RoboDK station: custom-palletizing.rdk

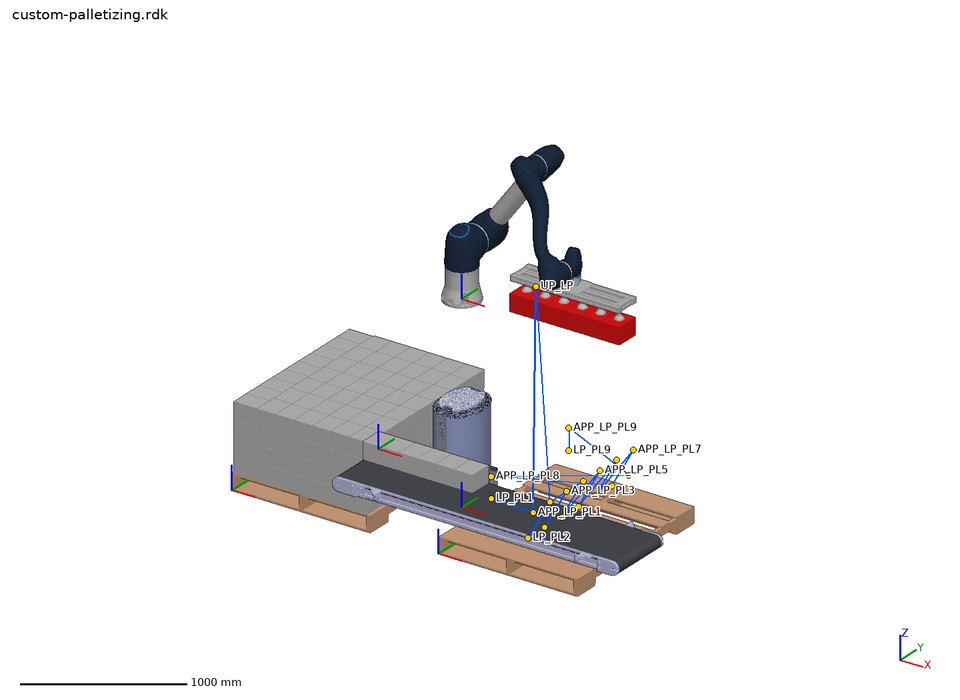
[picture v0: the station drawn from its stored meshes, robots at their saved joint values, targets as dots, program paths as lines]
Station custom-palletizing (saved by RoboDK 5.7.1). Poses are relative to the parent item; angles as X-Y-Z fixed-axis rotations.
Station parameters (name, value as stored): Conv_Run, 1
  - frame World at (0, 0, 0) mm
    - frame Doosan Robotics H2515 Base at (0, 0, 1390) mm
      - robot Doosan Robotics H2515: 6 axes, payload 25 kg, reach 1500 mm, repeatability 0.1 mm
          modified DH rows (alpha deg, a mm, theta deg, d mm): 0, 0, 0, 344.3; -90, 0, -90, -9.9; 0, 759.5, -90, 0; -90, 0, 0, 619.5; 90, 0, 0, 0; -90, 0, 0, 121
          base shift (0, 0, 0) mm, rotated rx 0 ry 0 rz 180 deg
          joint limits [-360, -130, -160, -360, -360, -360] to [360, 130, 160, 360, 360, 360]; home [0, 0, 90, 0, 0, 0]; saved at [0.72, 36.475, 109.267, -180, -34.248, -179.28]
        - tool Gripper, TCP at (0, 0, 145) mm, size 790 x 190 x 145 mm
          - object REF at (-402, -90, 0) mm, size 805 x 170 x 120 mm, geometry from 6 cajas.STEP
    - frame Conveyor_Frame at (0, -870, 737) mm
      - object Conveyor at (0, 300, -50) mm, size 2090.8 x 597 x 107.2 mm
      - object REF_CVY_BOX at (0, -170, 0) mm, size 805 x 170 x 120 mm, geometry from 6 cajas.STEP
      - folder Pick_poses
        - target APP_PICK (Cartesian target) at (402, -89.5, 320) mm, rotated rx 180 ry 0 rz 0 deg; joints [-67.813, 42.819, 79.411, 0, 57.77, 112.187] of Doosan Robotics H2515
        - target PICK_POSE (Cartesian target) at (402, -89.5, 120) mm, rotated rx -180 ry 0 rz 0 deg; joints [-67.813, 52.353, 82.536, 0, 45.111, 112.187] of Doosan Robotics H2515
        - target RET_PICK (Cartesian target) at (402, -89.5, 520) mm, rotated rx -180 ry 0 rz 0 deg; joints [-67.813, 36.264, 71.178, 0, 72.558, 112.187] of Doosan Robotics H2515
      - folder Pick_Aux_Poses
        - target UP_CONV (Cartesian target) at (402, 255, 850) mm, rotated rx -180 ry 0 rz 0 deg; joints [-57.601, 8.724, 80.723, 0, 90.554, 122.399] of Doosan Robotics H2515
    - frame Left_Pallet_Frame at (250, -600, 0) mm
      - object Left_Pallet at (0, 0, 0) mm, size 1016 x 1219.2 x 114.3 mm, geometry from Pallet-40x48in (1).sld
      - folder Ref_Box_LP
        - folder LAYER1
          - object REF_RP_BOX1 at (190, 0, 115) mm, size 805 x 170 x 120 mm, geometry from 6 cajas.STEP
          - object REF_RP_BOX2 at (190, 175, 115) mm, size 805 x 170 x 120 mm, geometry from 6 cajas.STEP
          - object REF_RP_BOX3 at (190, 350, 115) mm, size 805 x 170 x 120 mm, geometry from 6 cajas.STEP
          - object REF_RP_BOX4 at (190, 525, 115) mm, size 805 x 170 x 120 mm, geometry from 6 cajas.STEP
          - object REF_RP_BOX5 at (190, 700, 115) mm, size 805 x 170 x 120 mm, geometry from 6 cajas.STEP
          - object REF_RP_BOX6 at (190, 875, 115) mm, size 805 x 170 x 120 mm, geometry from 6 cajas.STEP
          - object REF_RP_BOX7 at (190, 1050, 115) mm, size 805 x 170 x 120 mm, geometry from 6 cajas.STEP
          - object REF_RP_BOX8 at (185, 0, 115) mm, rotated rx 0 ry 0 rz 90 deg, size 805 x 170 x 120 mm, geometry from 6 cajas.STEP
          - object REF_RP_BOX9 at (185, 810, 115) mm, rotated rx 0 ry 0 rz 90 deg, size 400 x 170 x 120 mm, geometry from 3 cajas.STEP
        - folder LAYER2
          - object REF_RP_BOX10 at (995, 815, 236) mm, rotated rx 0 ry 0 rz 90 deg, size 400 x 170 x 120 mm, geometry from 3 cajas.STEP
          - object REF_RP_BOX11 at (995, 5, 236) mm, rotated rx 0 ry 0 rz 90 deg, size 805 x 170 x 120 mm, geometry from 6 cajas.STEP
          - object REF_RP_BOX12 at (15, 0, 236) mm, size 805 x 170 x 120 mm, geometry from 6 cajas.STEP
          - object REF_RP_BOX13 at (15, 175, 236) mm, size 805 x 170 x 120 mm, geometry from 6 cajas.STEP
          - object REF_RP_BOX14 at (15, 350, 236) mm, size 805 x 170 x 120 mm, geometry from 6 cajas.STEP
          - object REF_RP_BOX15 at (15, 525, 236) mm, size 805 x 170 x 120 mm, geometry from 6 cajas.STEP
          - object REF_RP_BOX16 at (15, 700, 236) mm, size 805 x 170 x 120 mm, geometry from 6 cajas.STEP
          - object REF_RP_BOX17 at (15, 875, 236) mm, size 805 x 170 x 120 mm, geometry from 6 cajas.STEP
          - object REF_RP_BOX18 at (15, 1050, 236) mm, size 805 x 170 x 120 mm, geometry from 6 cajas.STEP
        - folder LAYER3
          - object REF_RP_BOX19 at (190, 0, 357) mm, size 805 x 170 x 120 mm, geometry from 6 cajas.STEP
          - object REF_RP_BOX20 at (190, 175, 357) mm, size 805 x 170 x 120 mm, geometry from 6 cajas.STEP
          - object REF_RP_BOX21 at (190, 350, 357) mm, size 805 x 170 x 120 mm, geometry from 6 cajas.STEP
          - object REF_RP_BOX22 at (190, 525, 357) mm, size 805 x 170 x 120 mm, geometry from 6 cajas.STEP
          - object REF_RP_BOX23 at (190, 700, 357) mm, size 805 x 170 x 120 mm, geometry from 6 cajas.STEP
          - object REF_RP_BOX24 at (190, 875, 357) mm, size 805 x 170 x 120 mm, geometry from 6 cajas.STEP
          - object REF_RP_BOX25 at (190, 1050, 357) mm, size 805 x 170 x 120 mm, geometry from 6 cajas.STEP
          - object REF_RP_BOX26 at (185, 0, 357) mm, rotated rx 0 ry 0 rz 90 deg, size 805 x 170 x 120 mm, geometry from 6 cajas.STEP
          - object REF_RP_BOX27 at (185, 810, 357) mm, rotated rx 0 ry 0 rz 90 deg, size 400 x 170 x 120 mm, geometry from 3 cajas.STEP
        - folder LAYER4
          - object REF_RP_BOX28 at (995, 815, 477) mm, rotated rx 0 ry 0 rz 90 deg, size 400 x 170 x 120 mm, geometry from 3 cajas.STEP
          - object REF_RP_BOX29 at (995, 5, 477) mm, rotated rx 0 ry 0 rz 90 deg, size 805 x 170 x 120 mm, geometry from 6 cajas.STEP
          - object REF_RP_BOX30 at (15, 0, 477) mm, size 805 x 170 x 120 mm, geometry from 6 cajas.STEP
          - object REF_RP_BOX31 at (15, 175, 477) mm, size 805 x 170 x 120 mm, geometry from 6 cajas.STEP
          - object REF_RP_BOX32 at (15, 350, 477) mm, size 805 x 170 x 120 mm, geometry from 6 cajas.STEP
          - object REF_RP_BOX33 at (15, 525, 477) mm, size 805 x 170 x 120 mm, geometry from 6 cajas.STEP
          - object REF_RP_BOX34 at (15, 700, 477) mm, size 805 x 170 x 120 mm, geometry from 6 cajas.STEP
          - object REF_RP_BOX35 at (15, 875, 477) mm, size 805 x 170 x 120 mm, geometry from 6 cajas.STEP
          - object REF_RP_BOX36 at (15, 1050, 477) mm, size 805 x 170 x 120 mm, geometry from 6 cajas.STEP
        - folder LAYER5
          - object REF_RP_BOX37 at (190, 0, 597) mm, size 805 x 170 x 120 mm, geometry from 6 cajas.STEP
          - object REF_RP_BOX38 at (190, 175, 597) mm, size 805 x 170 x 120 mm, geometry from 6 cajas.STEP
          - object REF_RP_BOX39 at (190, 350, 597) mm, size 805 x 170 x 120 mm, geometry from 6 cajas.STEP
          - object REF_RP_BOX40 at (190, 525, 597) mm, size 805 x 170 x 120 mm, geometry from 6 cajas.STEP
          - object REF_RP_BOX41 at (190, 700, 597) mm, size 805 x 170 x 120 mm, geometry from 6 cajas.STEP
          - object REF_RP_BOX42 at (190, 875, 597) mm, size 805 x 170 x 120 mm, geometry from 6 cajas.STEP
          - object REF_RP_BOX43 at (190, 1050, 597) mm, size 805 x 170 x 120 mm, geometry from 6 cajas.STEP
          - object REF_RP_BOX44 at (185, 0, 597) mm, rotated rx 0 ry 0 rz 90 deg, size 805 x 170 x 120 mm, geometry from 6 cajas.STEP
          - object REF_RP_BOX45 at (185, 810, 597) mm, rotated rx 0 ry 0 rz 90 deg, size 400 x 170 x 120 mm, geometry from 3 cajas.STEP
        - folder LAYER6
          - object REF_RP_BOX46 at (995, 815, 717) mm, rotated rx 0 ry 0 rz 90 deg, size 400 x 170 x 120 mm, geometry from 3 cajas.STEP
          - object REF_RP_BOX47 at (995, 5, 717) mm, rotated rx 0 ry 0 rz 90 deg, size 805 x 170 x 120 mm, geometry from 6 cajas.STEP
          - object REF_RP_BOX48 at (15, 0, 717) mm, size 805 x 170 x 120 mm, geometry from 6 cajas.STEP
          - object REF_RP_BOX49 at (15, 175, 717) mm, size 805 x 170 x 120 mm, geometry from 6 cajas.STEP
          - object REF_RP_BOX50 at (15, 350, 717) mm, size 805 x 170 x 120 mm, geometry from 6 cajas.STEP
          - object REF_RP_BOX51 at (15, 525, 717) mm, size 805 x 170 x 120 mm, geometry from 6 cajas.STEP
          - object REF_RP_BOX52 at (15, 700, 717) mm, size 805 x 170 x 120 mm, geometry from 6 cajas.STEP
          - object REF_RP_BOX53 at (15, 875, 717) mm, size 805 x 170 x 120 mm, geometry from 6 cajas.STEP
          - object REF_RP_BOX54 at (15, 1050, 717) mm, size 805 x 170 x 120 mm, geometry from 6 cajas.STEP
        - folder LAYER7
          - object REF_RP_BOX55 at (190, 0, 837) mm, size 805 x 170 x 120 mm, geometry from 6 cajas.STEP
          - object REF_RP_BOX56 at (190, 175, 837) mm, size 805 x 170 x 120 mm, geometry from 6 cajas.STEP
          - object REF_RP_BOX57 at (190, 350, 837) mm, size 805 x 170 x 120 mm, geometry from 6 cajas.STEP
          - object REF_RP_BOX58 at (190, 525, 837) mm, size 805 x 170 x 120 mm, geometry from 6 cajas.STEP
          - object REF_RP_BOX59 at (190, 700, 837) mm, size 805 x 170 x 120 mm, geometry from 6 cajas.STEP
          - object REF_RP_BOX60 at (190, 875, 837) mm, size 805 x 170 x 120 mm, geometry from 6 cajas.STEP
          - object REF_RP_BOX61 at (190, 1050, 837) mm, size 805 x 170 x 120 mm, geometry from 6 cajas.STEP
          - object REF_RP_BOX62 at (185, 0, 837) mm, rotated rx 0 ry 0 rz 90 deg, size 805 x 170 x 120 mm, geometry from 6 cajas.STEP
          - object REF_RP_BOX63 at (185, 810, 837) mm, rotated rx 0 ry 0 rz 90 deg, size 400 x 170 x 120 mm, geometry from 3 cajas.STEP
        - folder LAYER8
          - object REF_RP_BOX64 at (995, 815, 957) mm, rotated rx 0 ry 0 rz 90 deg, size 400 x 170 x 120 mm, geometry from 3 cajas.STEP
          - object REF_RP_BOX65 at (995, 5, 957) mm, rotated rx 0 ry 0 rz 90 deg, size 805 x 170 x 120 mm, geometry from 6 cajas.STEP
          - object REF_RP_BOX66 at (15, 0, 957) mm, size 805 x 170 x 120 mm, geometry from 6 cajas.STEP
          - object REF_RP_BOX67 at (15, 175, 957) mm, size 805 x 170 x 120 mm, geometry from 6 cajas.STEP
          - object REF_RP_BOX68 at (15, 350, 957) mm, size 805 x 170 x 120 mm, geometry from 6 cajas.STEP
          - object REF_RP_BOX69 at (15, 525, 957) mm, size 805 x 170 x 120 mm, geometry from 6 cajas.STEP
          - object REF_RP_BOX70 at (15, 700, 957) mm, size 805 x 170 x 120 mm, geometry from 6 cajas.STEP
          - object REF_RP_BOX71 at (15, 875, 957) mm, size 805 x 170 x 120 mm, geometry from 6 cajas.STEP
          - object REF_RP_BOX72 at (15, 1050, 957) mm, size 805 x 170 x 120 mm, geometry from 6 cajas.STEP
        - folder LAYER9
          - object REF_RP_BOX73 at (190, 0, 1077) mm, size 805 x 170 x 120 mm, geometry from 6 cajas.STEP
          - object REF_RP_BOX74 at (190, 175, 1077) mm, size 805 x 170 x 120 mm, geometry from 6 cajas.STEP
          - object REF_RP_BOX75 at (190, 350, 1077) mm, size 805 x 170 x 120 mm, geometry from 6 cajas.STEP
          - object REF_RP_BOX76 at (190, 525, 1077) mm, size 805 x 170 x 120 mm, geometry from 6 cajas.STEP
          - object REF_RP_BOX77 at (190, 700, 1077) mm, size 805 x 170 x 120 mm, geometry from 6 cajas.STEP
          - object REF_RP_BOX78 at (190, 875, 1077) mm, size 805 x 170 x 120 mm, geometry from 6 cajas.STEP
          - object REF_RP_BOX79 at (190, 1050, 1077) mm, size 805 x 170 x 120 mm, geometry from 6 cajas.STEP
          - object REF_RP_BOX80 at (185, 0, 1077) mm, rotated rx 0 ry 0 rz 90 deg, size 805 x 170 x 120 mm, geometry from 6 cajas.STEP
          - object REF_RP_BOX81 at (185, 810, 1077) mm, rotated rx 0 ry 0 rz 90 deg, size 400 x 170 x 120 mm, geometry from 3 cajas.STEP
      - folder LP_Aux_Poses
        - target UP_LP (Cartesian target) at (250, 660, 1590) mm, rotated rx 180 ry 0 rz 90 deg; joints [5.716, -8.781, 97.939, 0, 90.842, 95.716] of Doosan Robotics H2515
      - folder App_PL_LP
        - folder APP_LAYER 1
          - target APP_LP_PL1 (Cartesian target) at (593, 140, 385) mm, rotated rx -180 ry 0 rz -180 deg; joints [-29.211, 79.655, 80.222, 0, 20.123, -29.211] of Doosan Robotics H2515
          - target APP_LP_PL2 (Cartesian target) at (593, 315, 385) mm, rotated rx -180 ry 0 rz 180 deg; joints [-19.317, 78.101, 88.207, 0, 13.692, -19.317] of Doosan Robotics H2515
          - target APP_LP_PL3 (Cartesian target) at (593, 490, 385) mm, rotated rx -180 ry 0 rz -180 deg; joints [-8.102, 77.483, 92.417, 0, 10.1, -8.102] of Doosan Robotics H2515
          - target APP_LP_PL4 (Cartesian target) at (593, 665, 385) mm, rotated rx -180 ry 0 rz 180 deg; joints [3.738, 77.423, 92.897, 0, 9.68, 3.738] of Doosan Robotics H2515
          - target APP_LP_PL5 (Cartesian target) at (593, 840, 385) mm, rotated rx -180 ry 0 rz 180 deg; joints [15.244, 77.873, 89.645, 0, 12.482, 15.244] of Doosan Robotics H2515
          - target APP_LP_PL6 (Cartesian target) at (593, 1015, 385) mm, rotated rx -180 ry 0 rz -180 deg; joints [25.607, 79.136, 82.646, 0, 18.218, 25.607] of Doosan Robotics H2515
          - target APP_LP_PL7 (Cartesian target) at (593, 1190, 385) mm, rotated rx -180 ry 0 rz 180 deg; joints [34.436, 81.771, 71.646, 0, 26.584, 34.436] of Doosan Robotics H2515
          - target APP_LP_PL8 (Cartesian target) at (105, 402, 385) mm, rotated rx 180 ry 0 rz 90 deg; joints [-30.546, 85.041, 129.392, 0, -34.433, 59.454] of Doosan Robotics H2515
          - target APP_LP_PL9 (Cartesian target) at (105, 1212, 385) mm, rotated rx 180 ry 0 rz 90 deg; joints [59.082, 76.805, 106.157, 0, -2.962, 149.082] of Doosan Robotics H2515
        - folder APP_LAYER 2
          - target APP_LP_PL10 (Cartesian target) at (865, 812, 506) mm, rotated rx -180 ry 0 rz 90 deg; joints [9.768, 78.069, 62.913, 0, 39.018, 99.768] of Doosan Robotics H2515
          - target APP_LP_PL11 (Cartesian target) at (865, 407, 506) mm, rotated rx 180 ry 0 rz 90 deg; joints [-10.819, 78.078, 62.886, 0, 39.036, 79.181] of Doosan Robotics H2515
          - target APP_LP_PL12 (Cartesian target) at (418, 140, 506) mm, rotated rx 180 ry 0 rz 180 deg; joints [-35.824, 67.971, 101.551, 0, 10.478, -35.824] of Doosan Robotics H2515
          - target APP_LP_PL13 (Cartesian target) at (418, 315, 506) mm, rotated rx -180 ry 0 rz -180 deg; joints [-24.604, 67.188, 110.029, 0, 2.783, -24.604] of Doosan Robotics H2515
          - target APP_LP_PL14 (Cartesian target) at (418, 490, 506) mm, rotated rx -180 ry 0 rz -180 deg; joints [-11.02, 67.158, 114.814, 0, -1.972, -11.02] of Doosan Robotics H2515
          - target APP_LP_PL15 (Cartesian target) at (418, 665, 506) mm, rotated rx -180 ry 0 rz -180 deg; joints [3.861, 67.187, 115.58, 0, -2.766, 3.861] of Doosan Robotics H2515
          - target APP_LP_PL16 (Cartesian target) at (418, 840, 506) mm, rotated rx -180 ry 0 rz 180 deg; joints [18.196, 67.131, 112.257, 0, 0.612, 18.196] of Doosan Robotics H2515
          - target APP_LP_PL17 (Cartesian target) at (418, 1015, 506) mm, rotated rx 180 ry 0 rz 180 deg; joints [30.502, 67.544, 105.11, 0, 7.346, 30.502] of Doosan Robotics H2515
          - target APP_LP_PL18 (Cartesian target) at (418, 1190, 506) mm, rotated rx -180 ry 0 rz 180 deg; joints [40.325, 69.172, 94.445, 0, 16.383, 40.325] of Doosan Robotics H2515
        - folder APP_LAYER 3
          - target APP_LP_PL19 (Cartesian target) at (593, 140, 835) mm, rotated rx -180 ry 0 rz -180 deg; joints [-10.819, 78.078, 62.886, 0, 39.036, 79.181] of Doosan Robotics H2515
          - target APP_LP_PL20 (Cartesian target) at (593, 315, 835) mm, rotated rx -180 ry 0 rz 180 deg; joints [-10.819, 78.078, 62.886, 0, 39.036, 79.181] of Doosan Robotics H2515
          - target APP_LP_PL21 (Cartesian target) at (593, 490, 835) mm, rotated rx -180 ry 0 rz -180 deg; joints [-10.819, 78.078, 62.886, 0, 39.036, 79.181] of Doosan Robotics H2515
          - target APP_LP_PL22 (Cartesian target) at (593, 665, 835) mm, rotated rx -180 ry 0 rz 180 deg; joints [-10.819, 78.078, 62.886, 0, 39.036, 79.181] of Doosan Robotics H2515
          - target APP_LP_PL23 (Cartesian target) at (593, 840, 835) mm, rotated rx -180 ry 0 rz 180 deg; joints [-10.819, 78.078, 62.886, 0, 39.036, 79.181] of Doosan Robotics H2515
          - target APP_LP_PL24 (Cartesian target) at (593, 1015, 835) mm, rotated rx -180 ry 0 rz -180 deg; joints [-10.819, 78.078, 62.886, 0, 39.036, 79.181] of Doosan Robotics H2515
          - target APP_LP_PL25 (Cartesian target) at (593, 1190, 835) mm, rotated rx -180 ry 0 rz 180 deg; joints [-10.819, 78.078, 62.886, 0, 39.036, 79.181] of Doosan Robotics H2515
          - target APP_LP_PL26 (Cartesian target) at (105, 402, 835) mm, rotated rx 180 ry 0 rz 90 deg; joints [-10.819, 78.078, 62.886, 0, 39.036, 79.181] of Doosan Robotics H2515
          - target APP_LP_PL27 (Cartesian target) at (105, 1212, 835) mm, rotated rx 180 ry 0 rz 90 deg; joints [-10.819, 78.078, 62.886, 0, 39.036, 79.181] of Doosan Robotics H2515
        - folder APP_LAYER 4
          - target APP_LP_PL28 (Cartesian target) at (865, 812, 956) mm, rotated rx -180 ry 0 rz 90 deg; joints [-10.819, 78.078, 62.886, 0, 39.036, 79.181] of Doosan Robotics H2515
          - target APP_LP_PL29 (Cartesian target) at (865, 407, 956) mm, rotated rx 180 ry 0 rz 90 deg; joints [-10.819, 78.078, 62.886, 0, 39.036, 79.181] of Doosan Robotics H2515
          - target APP_LP_PL30 (Cartesian target) at (418, 140, 956) mm, rotated rx 180 ry 0 rz 180 deg; joints [-10.819, 78.078, 62.886, 0, 39.036, 79.181] of Doosan Robotics H2515
          - target APP_LP_PL31 (Cartesian target) at (418, 315, 956) mm, rotated rx -180 ry 0 rz -180 deg; joints [-10.819, 78.078, 62.886, 0, 39.036, 79.181] of Doosan Robotics H2515
          - target APP_LP_PL32 (Cartesian target) at (418, 490, 956) mm, rotated rx -180 ry 0 rz -180 deg; joints [-10.819, 78.078, 62.886, 0, 39.036, 79.181] of Doosan Robotics H2515
          - target APP_LP_PL33 (Cartesian target) at (418, 665, 956) mm, rotated rx -180 ry 0 rz -180 deg; joints [-10.819, 78.078, 62.886, 0, 39.036, 79.181] of Doosan Robotics H2515
          - target APP_LP_PL34 (Cartesian target) at (418, 840, 956) mm, rotated rx -180 ry 0 rz 180 deg; joints [-10.819, 78.078, 62.886, 0, 39.036, 79.181] of Doosan Robotics H2515
          - target APP_LP_PL35 (Cartesian target) at (418, 1015, 956) mm, rotated rx 180 ry 0 rz 180 deg; joints [-10.819, 78.078, 62.886, 0, 39.036, 79.181] of Doosan Robotics H2515
          - target APP_LP_PL36 (Cartesian target) at (418, 1190, 956) mm, rotated rx -180 ry 0 rz 180 deg; joints [-10.819, 78.078, 62.886, 0, 39.036, 79.181] of Doosan Robotics H2515
        - folder APP_LAYER 5
          - target APP_LP_PL37 (Cartesian target) at (593, 140, 1135) mm, rotated rx -180 ry 0 rz -180 deg; joints [-10.819, 78.078, 62.886, 0, 39.036, 79.181] of Doosan Robotics H2515
          - target APP_LP_PL38 (Cartesian target) at (593, 315, 1135) mm, rotated rx -180 ry 0 rz 180 deg; joints [-10.819, 78.078, 62.886, 0, 39.036, 79.181] of Doosan Robotics H2515
          - target APP_LP_PL39 (Cartesian target) at (593, 490, 1135) mm, rotated rx -180 ry 0 rz -180 deg; joints [-10.819, 78.078, 62.886, 0, 39.036, 79.181] of Doosan Robotics H2515
          - target APP_LP_PL40 (Cartesian target) at (593, 665, 1135) mm, rotated rx -180 ry 0 rz 180 deg; joints [-10.819, 78.078, 62.886, 0, 39.036, 79.181] of Doosan Robotics H2515
          - target APP_LP_PL41 (Cartesian target) at (593, 840, 1135) mm, rotated rx -180 ry 0 rz 180 deg; joints [-10.819, 78.078, 62.886, 0, 39.036, 79.181] of Doosan Robotics H2515
          - target APP_LP_PL42 (Cartesian target) at (593, 1015, 1135) mm, rotated rx -180 ry 0 rz -180 deg; joints [-10.819, 78.078, 62.886, 0, 39.036, 79.181] of Doosan Robotics H2515
          - target APP_LP_PL43 (Cartesian target) at (593, 1190, 1135) mm, rotated rx -180 ry 0 rz 180 deg; joints [-10.819, 78.078, 62.886, 0, 39.036, 79.181] of Doosan Robotics H2515
          - target APP_LP_PL44 (Cartesian target) at (105, 402, 1135) mm, rotated rx 180 ry 0 rz 90 deg; joints [-10.819, 78.078, 62.886, 0, 39.036, 79.181] of Doosan Robotics H2515
          - target APP_LP_PL45 (Cartesian target) at (105, 1212, 1135) mm, rotated rx 180 ry 0 rz 90 deg; joints [-10.819, 78.078, 62.886, 0, 39.036, 79.181] of Doosan Robotics H2515
        - folder APP_LAYER 6
          - target APP_LP_PL46 (Cartesian target) at (865, 812, 1256) mm, rotated rx -180 ry 0 rz 90 deg; joints [-10.819, 78.078, 62.886, 0, 39.036, 79.181] of Doosan Robotics H2515
          - target APP_LP_PL47 (Cartesian target) at (865, 407, 1256) mm, rotated rx 180 ry 0 rz 90 deg; joints [-10.819, 78.078, 62.886, 0, 39.036, 79.181] of Doosan Robotics H2515
          - target APP_LP_PL48 (Cartesian target) at (418, 140, 1256) mm, rotated rx 180 ry 0 rz 180 deg; joints [-10.819, 78.078, 62.886, 0, 39.036, 79.181] of Doosan Robotics H2515
          - target APP_LP_PL49 (Cartesian target) at (418, 315, 1256) mm, rotated rx -180 ry 0 rz -180 deg; joints [-10.819, 78.078, 62.886, 0, 39.036, 79.181] of Doosan Robotics H2515
          - target APP_LP_PL50 (Cartesian target) at (418, 490, 1256) mm, rotated rx -180 ry 0 rz -180 deg; joints [-10.819, 78.078, 62.886, 0, 39.036, 79.181] of Doosan Robotics H2515
          - target APP_LP_PL51 (Cartesian target) at (418, 665, 1256) mm, rotated rx -180 ry 0 rz -180 deg; joints [-10.819, 78.078, 62.886, 0, 39.036, 79.181] of Doosan Robotics H2515
          - target APP_LP_PL52 (Cartesian target) at (418, 840, 1256) mm, rotated rx -180 ry 0 rz 180 deg; joints [-10.819, 78.078, 62.886, 0, 39.036, 79.181] of Doosan Robotics H2515
          - target APP_LP_PL53 (Cartesian target) at (418, 1015, 1256) mm, rotated rx 180 ry 0 rz 180 deg; joints [-10.819, 78.078, 62.886, 0, 39.036, 79.181] of Doosan Robotics H2515
          - target APP_LP_PL54 (Cartesian target) at (418, 1190, 1256) mm, rotated rx -180 ry 0 rz 180 deg; joints [-10.819, 78.078, 62.886, 0, 39.036, 79.181] of Doosan Robotics H2515
        - folder APP_LAYER 7
          - target APP_LP_PL55 (Cartesian target) at (593, 140, 1435) mm, rotated rx -180 ry 0 rz -180 deg; joints [-10.819, 78.078, 62.886, 0, 39.036, 79.181] of Doosan Robotics H2515
          - target APP_LP_PL56 (Cartesian target) at (593, 315, 1435) mm, rotated rx -180 ry 0 rz 180 deg; joints [-10.819, 78.078, 62.886, 0, 39.036, 79.181] of Doosan Robotics H2515
          - target APP_LP_PL57 (Cartesian target) at (593, 490, 1435) mm, rotated rx -180 ry 0 rz -180 deg; joints [-10.819, 78.078, 62.886, 0, 39.036, 79.181] of Doosan Robotics H2515
          - target APP_LP_PL58 (Cartesian target) at (593, 665, 1435) mm, rotated rx -180 ry 0 rz 180 deg; joints [-10.819, 78.078, 62.886, 0, 39.036, 79.181] of Doosan Robotics H2515
          - target APP_LP_PL59 (Cartesian target) at (593, 840, 1435) mm, rotated rx -180 ry 0 rz 180 deg; joints [-10.819, 78.078, 62.886, 0, 39.036, 79.181] of Doosan Robotics H2515
          - target APP_LP_PL60 (Cartesian target) at (593, 1015, 1435) mm, rotated rx -180 ry 0 rz -180 deg; joints [-10.819, 78.078, 62.886, 0, 39.036, 79.181] of Doosan Robotics H2515
          - target APP_LP_PL61 (Cartesian target) at (593, 1190, 1435) mm, rotated rx -180 ry 0 rz 180 deg; joints [-10.819, 78.078, 62.886, 0, 39.036, 79.181] of Doosan Robotics H2515
          - target APP_LP_PL62 (Cartesian target) at (105, 402, 1435) mm, rotated rx 180 ry 0 rz 90 deg; joints [-10.819, 78.078, 62.886, 0, 39.036, 79.181] of Doosan Robotics H2515
          - target APP_LP_PL63 (Cartesian target) at (105, 1212, 1435) mm, rotated rx 180 ry 0 rz 90 deg; joints [-10.819, 78.078, 62.886, 0, 39.036, 79.181] of Doosan Robotics H2515
        - folder APP_LAYER 8
          - target APP_LP_PL64 (Cartesian target) at (865, 812, 1556) mm, rotated rx -180 ry 0 rz 90 deg; joints [-10.819, 78.078, 62.886, 0, 39.036, 79.181] of Doosan Robotics H2515
          - target APP_LP_PL65 (Cartesian target) at (865, 407, 1556) mm, rotated rx 180 ry 0 rz 90 deg; joints [-10.819, 78.078, 62.886, 0, 39.036, 79.181] of Doosan Robotics H2515
          - target APP_LP_PL66 (Cartesian target) at (418, 140, 1556) mm, rotated rx 180 ry 0 rz 180 deg; joints [-10.819, 78.078, 62.886, 0, 39.036, 79.181] of Doosan Robotics H2515
          - target APP_LP_PL67 (Cartesian target) at (418, 315, 1556) mm, rotated rx -180 ry 0 rz -180 deg; joints [-10.819, 78.078, 62.886, 0, 39.036, 79.181] of Doosan Robotics H2515
          - target APP_LP_PL68 (Cartesian target) at (418, 490, 1556) mm, rotated rx -180 ry 0 rz -180 deg; joints [-10.819, 78.078, 62.886, 0, 39.036, 79.181] of Doosan Robotics H2515
          - target APP_LP_PL69 (Cartesian target) at (418, 665, 1556) mm, rotated rx -180 ry 0 rz -180 deg; joints [-10.819, 78.078, 62.886, 0, 39.036, 79.181] of Doosan Robotics H2515
          - target APP_LP_PL70 (Cartesian target) at (418, 840, 1556) mm, rotated rx -180 ry 0 rz 180 deg; joints [-10.819, 78.078, 62.886, 0, 39.036, 79.181] of Doosan Robotics H2515
          - target APP_LP_PL71 (Cartesian target) at (418, 1015, 1556) mm, rotated rx 180 ry 0 rz 180 deg; joints [-10.819, 78.078, 62.886, 0, 39.036, 79.181] of Doosan Robotics H2515
          - target APP_LP_PL72 (Cartesian target) at (418, 1190, 1556) mm, rotated rx -180 ry 0 rz 180 deg; joints [-10.819, 78.078, 62.886, 0, 39.036, 79.181] of Doosan Robotics H2515
        - folder APP_LAYER 9
          - target APP_LP_PL73 (Cartesian target) at (593, 140, 1735) mm, rotated rx -180 ry 0 rz -180 deg; joints [-10.819, 78.078, 62.886, 0, 39.036, 79.181] of Doosan Robotics H2515
          - target APP_LP_PL74 (Cartesian target) at (593, 315, 1735) mm, rotated rx -180 ry 0 rz 180 deg; joints [-10.819, 78.078, 62.886, 0, 39.036, 79.181] of Doosan Robotics H2515
          - target APP_LP_PL75 (Cartesian target) at (593, 490, 1735) mm, rotated rx -180 ry 0 rz -180 deg; joints [-10.819, 78.078, 62.886, 0, 39.036, 79.181] of Doosan Robotics H2515
          - target APP_LP_PL76 (Cartesian target) at (593, 665, 1735) mm, rotated rx -180 ry 0 rz 180 deg; joints [-10.819, 78.078, 62.886, 0, 39.036, 79.181] of Doosan Robotics H2515
          - target APP_LP_PL77 (Cartesian target) at (593, 840, 1735) mm, rotated rx -180 ry 0 rz 180 deg; joints [-10.819, 78.078, 62.886, 0, 39.036, 79.181] of Doosan Robotics H2515
          - target APP_LP_PL78 (Cartesian target) at (593, 1015, 1735) mm, rotated rx -180 ry 0 rz -180 deg; joints [-10.819, 78.078, 62.886, 0, 39.036, 79.181] of Doosan Robotics H2515
          - target APP_LP_PL79 (Cartesian target) at (593, 1190, 1735) mm, rotated rx -180 ry 0 rz 180 deg; joints [-10.819, 78.078, 62.886, 0, 39.036, 79.181] of Doosan Robotics H2515
          - target APP_LP_PL80 (Cartesian target) at (105, 402, 1735) mm, rotated rx 180 ry 0 rz 90 deg; joints [-10.819, 78.078, 62.886, 0, 39.036, 79.181] of Doosan Robotics H2515
          - target APP_LP_PL81 (Cartesian target) at (105, 1212, 1735) mm, rotated rx 180 ry 0 rz 90 deg; joints [-10.819, 78.078, 62.886, 0, 39.036, 79.181] of Doosan Robotics H2515
      - folder Place_LP
        - folder PL_LAYER 1
          - target LP_PL1 (Cartesian target) at (105, 402, 235) mm, rotated rx 180 ry 0 rz 90 deg; joints [-30.546, 96.287, 117.953, 0, -34.24, 59.454] of Doosan Robotics H2515
          - target LP_PL2 (Cartesian target) at (593, 90, 235) mm, rotated rx -180 ry 0 rz 180 deg; joints [-31.749, 91.394, 67.216, 0, 21.39, -31.749] of Doosan Robotics H2515
          - target LP_PL3 (Cartesian target) at (593, 265, 235) mm, rotated rx -180 ry 0 rz 180 deg; joints [-22.298, 89.52, 76.696, 0, 13.783, -22.298] of Doosan Robotics H2515
          - target LP_PL4 (Cartesian target) at (593, 440, 235) mm, rotated rx -180 ry 0 rz 180 deg; joints [-11.408, 88.771, 82.065, 0, 9.164, -11.408] of Doosan Robotics H2515
          - target LP_PL5 (Cartesian target) at (593, 615, 235) mm, rotated rx -180 ry 0 rz -180 deg; joints [0.347, 88.604, 83.622, 0, 7.774, 0.347] of Doosan Robotics H2515
          - target LP_PL6 (Cartesian target) at (593, 790, 235) mm, rotated rx -180 ry 0 rz 180 deg; joints [12.045, 88.847, 81.419, 0, 9.734, 12.045] of Doosan Robotics H2515
          - target LP_PL7 (Cartesian target) at (593, 965, 235) mm, rotated rx -180 ry 0 rz -180 deg; joints [22.794, 89.741, 75.379, 0, 14.88, 22.794] of Doosan Robotics H2515
          - target LP_PL8 (Cartesian target) at (593, 1140, 235) mm, rotated rx -180 ry 0 rz 180 deg; joints [32.076, 91.888, 65.12, 0, 22.993, 32.076] of Doosan Robotics H2515
          - target LP_PL9 (Cartesian target) at (105, 1212, 235) mm, rotated rx 180 ry 0 rz 90 deg; joints [59.082, 88.337, 96.453, 0, -4.791, 149.082] of Doosan Robotics H2515
        - folder PL_LAYER 2
          - target LP_PL10 (Cartesian target) at (915, 812, 356) mm, rotated rx -180 ry 0 rz 90 deg; joints [9.357, 91.648, 45.269, 0, 43.083, 99.357] of Doosan Robotics H2515
          - target LP_PL11 (Cartesian target) at (915, 407, 356) mm, rotated rx -180 ry 0 rz 90 deg; joints [-10.364, 91.66, 45.234, 0, 43.105, 79.636] of Doosan Robotics H2515
          - target LP_PL12 (Cartesian target) at (418, 90, 356) mm, rotated rx -180 ry 0 rz -180 deg; joints [-38.569, 79.596, 91.165, 0, 9.239, -38.569] of Doosan Robotics H2515
          - target LP_PL13 (Cartesian target) at (418, 265, 356) mm, rotated rx 180 ry 0 rz 180 deg; joints [-28.069, 78.981, 100.439, 0, 0.58, -28.069] of Doosan Robotics H2515
          - target LP_PL14 (Cartesian target) at (418, 440, 356) mm, rotated rx -180 ry 0 rz 180 deg; joints [-15.101, 79.179, 106.079, 0, -5.258, -15.101] of Doosan Robotics H2515
          - target LP_PL15 (Cartesian target) at (418, 615, 356) mm, rotated rx -180 ry 0 rz 180 deg; joints [-0.42, 79.362, 107.918, 0, -7.28, -0.42] of Doosan Robotics H2515
          - target LP_PL16 (Cartesian target) at (418, 790, 356) mm, rotated rx -180 ry 0 rz 180 deg; joints [14.261, 79.161, 105.858, 0, -5.019, 14.261] of Doosan Robotics H2515
          - target LP_PL17 (Cartesian target) at (418, 965, 356) mm, rotated rx 180 ry 0 rz 180 deg; joints [27.238, 78.986, 100.006, 0, 1.008, 27.238] of Doosan Robotics H2515
          - target LP_PL18 (Cartesian target) at (418, 1140, 356) mm, rotated rx -180 ry 0 rz 180 deg; joints [37.764, 79.673, 90.526, 0, 9.802, 37.764] of Doosan Robotics H2515
        - folder PL_LAYER 3
          - target LP_PL19 (Cartesian target) at (105, 402, 477) mm, rotated rx 180 ry 0 rz 90 deg; joints [-30.546, 75.175, 136.778, -180, 31.953, -120.546] of Doosan Robotics H2515
          - target LP_PL20 (Cartesian target) at (593, 90, 477) mm, rotated rx -180 ry 0 rz 180 deg; joints [-31.749, 72.348, 82.687, 0, 24.966, -31.749] of Doosan Robotics H2515
          - target LP_PL21 (Cartesian target) at (593, 265, 477) mm, rotated rx -180 ry 0 rz -180 deg; joints [-22.298, 70.181, 91.71, -180, -18.109, -202.298] of Doosan Robotics H2515
          - target LP_PL22 (Cartesian target) at (593, 440, 477) mm, rotated rx -180 ry 0 rz -180 deg; joints [-11.408, 69.159, 97.002, -180, -13.84, -191.408] of Doosan Robotics H2515
          - target LP_PL23 (Cartesian target) at (593, 615, 477) mm, rotated rx -180 ry 0 rz -180 deg; joints [0.347, 68.9, 98.561, -180, -12.539, -179.653] of Doosan Robotics H2515
          - target LP_PL24 (Cartesian target) at (593, 790, 477) mm, rotated rx -180 ry 0 rz -180 deg; joints [12.045, 69.272, 96.358, -180, -14.37, -167.955] of Doosan Robotics H2515
          - target LP_PL25 (Cartesian target) at (593, 965, 477) mm, rotated rx -180 ry 0 rz -180 deg; joints [22.794, 70.458, 90.431, -180, -19.111, -157.206] of Doosan Robotics H2515
          - target LP_PL26 (Cartesian target) at (593, 1140, 477) mm, rotated rx 180 ry 0 rz 180 deg; joints [32.076, 72.871, 80.748, -180, -26.38, -147.924] of Doosan Robotics H2515
          - target LP_PL27 (Cartesian target) at (105, 1212, 477) mm, rotated rx 180 ry 0 rz 90 deg; joints [59.082, 67.701, 111.861, 0, 0.438, -210.918] of Doosan Robotics H2515
        - folder PL_LAYER 4
          - target LP_PL28 (Cartesian target) at (915, 812, 597) mm, rotated rx -180 ry 0 rz 90 deg; joints [9.834, 73.95, 58.898, 0, 47.153, 99.834] of Doosan Robotics H2515
          - target LP_PL29 (Cartesian target) at (915, 407, 597) mm, rotated rx -180 ry 0 rz 90 deg; joints [-9.887, 73.741, 59.444, 0, 46.816, 80.113] of Doosan Robotics H2515
          - target LP_PL30 (Cartesian target) at (418, 90, 597) mm, rotated rx -180 ry 0 rz -180 deg; joints [-38.036, 59.932, 102.879, 0, 17.189, -38.036] of Doosan Robotics H2515
          - target LP_PL31 (Cartesian target) at (418, 265, 597) mm, rotated rx -180 ry 0 rz 180 deg; joints [-27.393, 58.235, 112.336, 0, 9.429, -27.393] of Doosan Robotics H2515
          - target LP_PL32 (Cartesian target) at (418, 440, 597) mm, rotated rx -180 ry 0 rz -180 deg; joints [-14.296, 57.637, 118.17, 0, 4.193, -14.296] of Doosan Robotics H2515
          - target LP_PL33 (Cartesian target) at (418, 615, 597) mm, rotated rx -180 ry 0 rz -180 deg; joints [0.437, 57.543, 119.938, 0, 2.52, 0.437] of Doosan Robotics H2515
          - target LP_PL34 (Cartesian target) at (418, 790, 597) mm, rotated rx -180 ry 0 rz -180 deg; joints [15.061, 57.689, 117.447, 0, 4.864, 15.061] of Doosan Robotics H2515
          - target LP_PL35 (Cartesian target) at (418, 965, 597) mm, rotated rx 180 ry 0 rz -180 deg; joints [27.907, 58.431, 110.96, 0, 10.608, 27.907] of Doosan Robotics H2515
          - target LP_PL36 (Cartesian target) at (418, 1140, 597) mm, rotated rx -180 ry 0 rz -180 deg; joints [38.291, 60.372, 100.919, 0, 18.709, 38.291] of Doosan Robotics H2515
        - folder PL_LAYER 5
          - target LP_PL37 (Cartesian target) at (105, 402, 717) mm, rotated rx 180 ry 0 rz 90 deg; joints [-30.546, 48.067, 146.771, -180, 14.839, -120.546] of Doosan Robotics H2515
          - target LP_PL38 (Cartesian target) at (593, 90, 717) mm, rotated rx -180 ry 0 rz 180 deg; joints [-31.749, 56.539, 88.882, 0, 34.579, -31.749] of Doosan Robotics H2515
          - target LP_PL39 (Cartesian target) at (593, 265, 717) mm, rotated rx -180 ry 0 rz -180 deg; joints [-22.298, 53.443, 97.91, -180, -28.646, -202.298] of Doosan Robotics H2515
          - target LP_PL40 (Cartesian target) at (593, 440, 717) mm, rotated rx 180 ry 0 rz -180 deg; joints [-11.408, 51.744, 103.278, 0, 24.977, -11.408] of Doosan Robotics H2515
          - target LP_PL41 (Cartesian target) at (593, 615, 717) mm, rotated rx -180 ry 0 rz 180 deg; joints [0.347, 51.265, 104.871, -180, -23.864, -179.653] of Doosan Robotics H2515
          - target LP_PL42 (Cartesian target) at (593, 790, 717) mm, rotated rx 180 ry 0 rz -180 deg; joints [12.045, 51.945, 102.622, -180, -25.432, -167.955] of Doosan Robotics H2515
          - target LP_PL43 (Cartesian target) at (593, 965, 717) mm, rotated rx -180 ry 0 rz 180 deg; joints [22.794, 53.868, 96.621, -180, -29.51, -157.206] of Doosan Robotics H2515
          - target LP_PL44 (Cartesian target) at (593, 1140, 717) mm, rotated rx 180 ry 0 rz 180 deg; joints [32.076, 57.229, 86.962, -180, -35.808, -147.924] of Doosan Robotics H2515
          - target LP_PL45 (Cartesian target) at (105, 1212, 717) mm, rotated rx 180 ry 0 rz 90 deg; joints [59.082, 47.727, 118.694, 0, 13.579, -210.918] of Doosan Robotics H2515
        - folder PL_LAYER 6
          - target LP_PL46 (Cartesian target) at (915, 812, 837) mm, rotated rx -180 ry 0 rz 90 deg; joints [9.834, 80.867, 54.632, -180, -44.501, -80.166] of Doosan Robotics H2515
          - target LP_PL47 (Cartesian target) at (915, 407, 837) mm, rotated rx 180 ry 0 rz 90 deg; joints [-9.887, 80.657, 55.205, -180, -44.138, -99.887] of Doosan Robotics H2515
          - target LP_PL48 (Cartesian target) at (418, 90, 837) mm, rotated rx -180 ry 0 rz -180 deg; joints [-38.036, 68.109, 99.244, -180, -12.647, -218.036] of Doosan Robotics H2515
          - target LP_PL49 (Cartesian target) at (418, 265, 837) mm, rotated rx 180 ry 0 rz -180 deg; joints [-27.393, 67.034, 108.529, -180, -4.437, -207.393] of Doosan Robotics H2515
          - target LP_PL50 (Cartesian target) at (418, 440, 837) mm, rotated rx 180 ry 0 rz 180 deg; joints [-14.296, 66.891, 114.194, -180, 1.085, -194.296] of Doosan Robotics H2515
          - target LP_PL51 (Cartesian target) at (418, 615, 837) mm, rotated rx -180 ry 0 rz 180 deg; joints [0.437, 66.945, 115.9, -180, 2.844, -179.563] of Doosan Robotics H2515
          - target LP_PL52 (Cartesian target) at (418, 790, 837) mm, rotated rx -180 ry 0 rz 180 deg; joints [15.061, 66.883, 113.495, -180, 0.378, -164.939] of Doosan Robotics H2515
          - target LP_PL53 (Cartesian target) at (418, 965, 837) mm, rotated rx -180 ry 0 rz -180 deg; joints [27.907, 67.132, 107.185, -180, -5.683, -152.093] of Doosan Robotics H2515
          - target LP_PL54 (Cartesian target) at (418, 1140, 837) mm, rotated rx 180 ry 0 rz 180 deg; joints [38.291, 68.438, 97.306, -180, -14.256, -141.709] of Doosan Robotics H2515
        - folder PL_LAYER 7
          - target LP_PL55 (Cartesian target) at (105, 402, 957) mm, rotated rx 180 ry 0 rz 90 deg; joints [-30.546, 61.719, 143.349, -180, 25.068, -120.546] of Doosan Robotics H2515
          - target LP_PL56 (Cartesian target) at (593, 90, 957) mm, rotated rx -180 ry 0 rz 180 deg; joints [-31.749, 63.583, 86.921, -180, -29.497, -211.749] of Doosan Robotics H2515
          - target LP_PL57 (Cartesian target) at (593, 265, 957) mm, rotated rx -180 ry 0 rz 180 deg; joints [-22.298, 60.97, 95.936, -180, -23.093, -202.298] of Doosan Robotics H2515
          - target LP_PL58 (Cartesian target) at (593, 440, 957) mm, rotated rx -180 ry 0 rz -180 deg; joints [-11.408, 59.622, 101.273, -180, -19.105, -191.408] of Doosan Robotics H2515
          - target LP_PL59 (Cartesian target) at (593, 615, 957) mm, rotated rx -180 ry 0 rz -180 deg; joints [0.347, 59.257, 102.853, -180, -17.89, -179.653] of Doosan Robotics H2515
          - target LP_PL60 (Cartesian target) at (593, 790, 957) mm, rotated rx -180 ry 0 rz 180 deg; joints [12.045, 59.778, 100.621, -180, -19.601, -167.955] of Doosan Robotics H2515
          - target LP_PL61 (Cartesian target) at (593, 965, 957) mm, rotated rx 180 ry 0 rz 180 deg; joints [22.794, 61.319, 94.652, -180, -24.029, -157.206] of Doosan Robotics H2515
          - target LP_PL62 (Cartesian target) at (593, 1140, 957) mm, rotated rx 180 ry 0 rz 180 deg; joints [32.076, 64.185, 84.998, -180, -30.817, -147.924] of Doosan Robotics H2515
          - target LP_PL63 (Cartesian target) at (105, 1212, 957) mm, rotated rx 180 ry 0 rz 90 deg; joints [59.082, 56.956, 116.483, -180, -6.561, -30.918] of Doosan Robotics H2515
        - folder PL_LAYER 8
          - target LP_PL64 (Cartesian target) at (915, 812, 1077) mm, rotated rx 180 ry 0 rz 90 deg; joints [9.834, 66.606, 61.566, -180, -51.828, -80.166] of Doosan Robotics H2515
          - target LP_PL65 (Cartesian target) at (915, 407, 1077) mm, rotated rx 180 ry 0 rz 90 deg; joints [-9.887, 66.387, 62.098, -180, -51.515, -99.887] of Doosan Robotics H2515
          - target LP_PL66 (Cartesian target) at (418, 90, 1077) mm, rotated rx -180 ry 0 rz 180 deg; joints [-38.036, 50.465, 105.267, -180, -24.268, -218.036] of Doosan Robotics H2515
          - target LP_PL67 (Cartesian target) at (418, 265, 1077) mm, rotated rx -180 ry 0 rz -180 deg; joints [-27.393, 47.809, 114.864, -180, -17.328, -207.393] of Doosan Robotics H2515
          - target LP_PL68 (Cartesian target) at (418, 440, 1077) mm, rotated rx -180 ry 0 rz -180 deg; joints [-14.296, 46.474, 120.831, -180, -12.695, -194.296] of Doosan Robotics H2515
          - target LP_PL69 (Cartesian target) at (418, 615, 1077) mm, rotated rx -180 ry 0 rz -180 deg; joints [0.437, 46.13, 122.648, -180, -11.222, -179.563] of Doosan Robotics H2515
          - target LP_PL70 (Cartesian target) at (418, 790, 1077) mm, rotated rx -180 ry 0 rz 180 deg; joints [15.061, 46.623, 120.09, -180, -13.287, -164.939] of Doosan Robotics H2515
          - target LP_PL71 (Cartesian target) at (418, 965, 1077) mm, rotated rx 180 ry 0 rz 180 deg; joints [27.907, 48.162, 113.462, -180, -18.376, -152.093] of Doosan Robotics H2515
          - target LP_PL72 (Cartesian target) at (418, 1140, 1077) mm, rotated rx 180 ry 0 rz 180 deg; joints [38.291, 51.074, 103.288, -180, -25.638, -141.709] of Doosan Robotics H2515
        - folder PL_LAYER 9
          - target LP_PL73 (Cartesian target) at (105, 402, 1197) mm, rotated rx 180 ry 0 rz 90 deg; joints [-30.546, 30.017, 147.539, -180, -2.444, -120.546] of Doosan Robotics H2515
          - target LP_PL74 (Cartesian target) at (593, 90, 1197) mm, rotated rx 180 ry 0 rz 180 deg; joints [-31.749, 48.828, 89.298, -180, -41.874, -211.749] of Doosan Robotics H2515
          - target LP_PL75 (Cartesian target) at (593, 265, 1197) mm, rotated rx -180 ry 0 rz -180 deg; joints [-22.298, 45.091, 98.331, -180, -36.578, -202.298] of Doosan Robotics H2515
          - target LP_PL76 (Cartesian target) at (593, 440, 1197) mm, rotated rx -180 ry 0 rz -180 deg; joints [-11.408, 42.929, 103.706, -180, -33.364, -191.408] of Doosan Robotics H2515
          - target LP_PL77 (Cartesian target) at (593, 615, 1197) mm, rotated rx -180 ry 0 rz 180 deg; joints [0.347, 42.298, 105.302, -180, -32.399, -179.653] of Doosan Robotics H2515
          - target LP_PL78 (Cartesian target) at (593, 790, 1197) mm, rotated rx 180 ry 0 rz 180 deg; joints [12.045, 43.191, 103.049, -180, -33.76, -167.955] of Doosan Robotics H2515
          - target LP_PL79 (Cartesian target) at (593, 965, 1197) mm, rotated rx -180 ry 0 rz 180 deg; joints [22.794, 45.618, 97.041, -180, -37.341, -157.206] of Doosan Robotics H2515
          - target LP_PL80 (Cartesian target) at (593, 1140, 1197) mm, rotated rx 180 ry 0 rz 180 deg; joints [32.076, 49.636, 87.379, -180, -42.985, -147.924] of Doosan Robotics H2515
          - target LP_PL81 (Cartesian target) at (105, 1212, 1197) mm, rotated rx 180 ry 0 rz 90 deg; joints [59.082, 37.095, 119.17, -180, -23.735, -30.918] of Doosan Robotics H2515
      - folder Waypoints_LP
        - target MID_LP_L1 (Cartesian target) at (550, 620, 600) mm, rotated rx -180 ry 0 rz -180 deg; joints [0.723, 58.862, 107.115, 0, 14.023, 0.723] of Doosan Robotics H2515
        - target MID_LP_L2 (Cartesian target) at (550, 620, 721) mm, rotated rx -180 ry 0 rz -180 deg; joints [0.723, 49.683, 109.408, 0, 20.909, 0.723] of Doosan Robotics H2515
        - target MID_LP_L3 (Cartesian target) at (550, 620, 842) mm, rotated rx -180 ry 0 rz -180 deg; joints [0.723, 40.898, 109.827, 0, 29.274, 0.723] of Doosan Robotics H2515
        - target MID_LP_L4 (Cartesian target) at (550, 620, 962) mm, rotated rx -180 ry 0 rz -180 deg; joints [0.723, 32.947, 108.378, 0, 38.674, 0.723] of Doosan Robotics H2515
        - target MID_LP_L5 (Cartesian target) at (550, 620, 1082) mm, rotated rx -180 ry 0 rz -180 deg; joints [0.723, 26.111, 105.117, 0, 48.772, 0.723] of Doosan Robotics H2515
      - target Target 169 (Cartesian target) at (550.09, 619.96, 1087) mm, rotated rx -180 ry 0.01 rz -180 deg; joints [0.72, 52.239, 108.947, 0, 18.805, 0.72] of Doosan Robotics H2515
      - target Target 170 (Cartesian target) at (550.09, 619.96, 1207) mm, rotated rx 180 ry 0.01 rz -180 deg; joints [0.72, 43.379, 109.896, 0, 26.715, 0.72] of Doosan Robotics H2515
      - target Target 171 (Cartesian target) at (550.09, 619.96, 1327) mm, rotated rx 180 ry 0.01 rz -180 deg; joints [0.72, 35.168, 108.987, 0, 35.835, 0.72] of Doosan Robotics H2515
      - target Target 172 (Cartesian target) at (550.09, 619.96, 1447) mm, rotated rx 180 ry 0.01 rz -180 deg; joints [0.72, 27.974, 106.247, 0, 45.769, 0.72] of Doosan Robotics H2515
      - target Target 173 (Cartesian target) at (550.09, 619.96, 1567) mm, rotated rx -180 ry 0.01 rz -180 deg; joints [0.72, 22.096, 101.747, 0, 56.146, 0.72] of Doosan Robotics H2515
    - frame Right_Pallet_Frame at (-1266, -600, 0) mm
      - object Right_Pallet at (0, 0, 0) mm, size 1016 x 1219.2 x 114.3 mm, geometry from Pallet-40x48in (1).sld
      - folder Ref_Box_RP
        - folder LAYER 1
          - object REF_RP_BOX1 at (995, 0, 115) mm, rotated rx 0 ry 0 rz 90 deg, size 805 x 170 x 120 mm, geometry from 6 cajas.STEP
          - object REF_RP_BOX2 at (15, 0, 115) mm, size 805 x 170 x 120 mm, geometry from 6 cajas.STEP
          - object REF_RP_BOX3 at (15, 175, 115) mm, size 805 x 170 x 120 mm, geometry from 6 cajas.STEP
          - object REF_RP_BOX4 at (15, 350, 115) mm, size 805 x 170 x 120 mm, geometry from 6 cajas.STEP
          - object REF_RP_BOX5 at (15, 525, 115) mm, size 805 x 170 x 120 mm, geometry from 6 cajas.STEP
          - object REF_RP_BOX6 at (15, 700, 115) mm, size 805 x 170 x 120 mm, geometry from 6 cajas.STEP
          - object REF_RP_BOX7 at (15, 875, 115) mm, size 805 x 170 x 120 mm, geometry from 6 cajas.STEP
          - object REF_RP_BOX8 at (15, 1050, 115) mm, size 805 x 170 x 120 mm, geometry from 6 cajas.STEP
          - object REF_RP_BOX9 at (995, 810, 115) mm, rotated rx 0 ry 0 rz 90 deg, size 400 x 170 x 120 mm, geometry from 3 cajas.STEP
        - folder LAYER 2
          - object REF_RP_BOX10 at (185, 810, 236) mm, rotated rx 0 ry 0 rz 90 deg, size 400 x 170 x 120 mm, geometry from 3 cajas.STEP
          - object REF_RP_BOX11 at (185, 0, 236) mm, rotated rx 0 ry 0 rz 90 deg, size 805 x 170 x 120 mm, geometry from 6 cajas.STEP
          - object REF_RP_BOX12 at (191, 0, 236) mm, size 805 x 170 x 120 mm, geometry from 6 cajas.STEP
          - object REF_RP_BOX13 at (191, 175, 236) mm, size 805 x 170 x 120 mm, geometry from 6 cajas.STEP
          - object REF_RP_BOX14 at (191, 350, 236) mm, size 805 x 170 x 120 mm, geometry from 6 cajas.STEP
          - object REF_RP_BOX15 at (191, 525, 236) mm, size 805 x 170 x 120 mm, geometry from 6 cajas.STEP
          - object REF_RP_BOX16 at (191, 700, 236) mm, size 805 x 170 x 120 mm, geometry from 6 cajas.STEP
          - object REF_RP_BOX17 at (191, 875, 236) mm, size 805 x 170 x 120 mm, geometry from 6 cajas.STEP
          - object REF_RP_BOX18 at (191, 1050, 236) mm, size 805 x 170 x 120 mm, geometry from 6 cajas.STEP
        - folder LAYER 3
          - object REF_RP_BOX19 at (995, 0, 357) mm, rotated rx 0 ry 0 rz 90 deg, size 805 x 170 x 120 mm, geometry from 6 cajas.STEP
          - object REF_RP_BOX20 at (15, 0, 357) mm, size 805 x 170 x 120 mm, geometry from 6 cajas.STEP
          - object REF_RP_BOX21 at (15, 175, 357) mm, size 805 x 170 x 120 mm, geometry from 6 cajas.STEP
          - object REF_RP_BOX22 at (15, 350, 357) mm, size 805 x 170 x 120 mm, geometry from 6 cajas.STEP
          - object REF_RP_BOX23 at (15, 525, 357) mm, size 805 x 170 x 120 mm, geometry from 6 cajas.STEP
          - object REF_RP_BOX24 at (15, 700, 357) mm, size 805 x 170 x 120 mm, geometry from 6 cajas.STEP
          - object REF_RP_BOX25 at (15, 875, 357) mm, size 805 x 170 x 120 mm, geometry from 6 cajas.STEP
          - object REF_RP_BOX26 at (15, 1050, 357) mm, size 805 x 170 x 120 mm, geometry from 6 cajas.STEP
          - object REF_RP_BOX27 at (995, 810, 357) mm, rotated rx 0 ry 0 rz 90 deg, size 400 x 170 x 120 mm, geometry from 3 cajas.STEP
        - folder LAYER 4
          - object REF_RP_BOX28 at (185, 810, 478) mm, rotated rx 0 ry 0 rz 90 deg, size 400 x 170 x 120 mm, geometry from 3 cajas.STEP
          - object REF_RP_BOX29 at (185, 0, 478) mm, rotated rx 0 ry 0 rz 90 deg, size 805 x 170 x 120 mm, geometry from 6 cajas.STEP
          - object REF_RP_BOX30 at (191, 0, 478) mm, size 805 x 170 x 120 mm, geometry from 6 cajas.STEP
          - object REF_RP_BOX31 at (191, 175, 478) mm, size 805 x 170 x 120 mm, geometry from 6 cajas.STEP
          - object REF_RP_BOX32 at (191, 350, 478) mm, size 805 x 170 x 120 mm, geometry from 6 cajas.STEP
          - object REF_RP_BOX33 at (191, 525, 478) mm, size 805 x 170 x 120 mm, geometry from 6 cajas.STEP
          - object REF_RP_BOX34 at (191, 700, 478) mm, size 805 x 170 x 120 mm, geometry from 6 cajas.STEP
          - object REF_RP_BOX35 at (191, 875, 478) mm, size 805 x 170 x 120 mm, geometry from 6 cajas.STEP
          - object REF_RP_BOX36 at (191, 1050, 478) mm, size 805 x 170 x 120 mm, geometry from 6 cajas.STEP
        - folder LAYER 5
          - object REF_RP_BOX37 at (995, 0, 599) mm, rotated rx 0 ry 0 rz 90 deg, size 805 x 170 x 120 mm, geometry from 6 cajas.STEP
          - object REF_RP_BOX38 at (15, 0, 599) mm, size 805 x 170 x 120 mm, geometry from 6 cajas.STEP
          - object REF_RP_BOX39 at (15, 175, 599) mm, size 805 x 170 x 120 mm, geometry from 6 cajas.STEP
          - object REF_RP_BOX40 at (15, 350, 599) mm, size 805 x 170 x 120 mm, geometry from 6 cajas.STEP
          - object REF_RP_BOX41 at (15, 525, 599) mm, size 805 x 170 x 120 mm, geometry from 6 cajas.STEP
          - object REF_RP_BOX42 at (15, 700, 599) mm, size 805 x 170 x 120 mm, geometry from 6 cajas.STEP
          - object REF_RP_BOX43 at (15, 875, 599) mm, size 805 x 170 x 120 mm, geometry from 6 cajas.STEP
          - object REF_RP_BOX44 at (15, 1050, 599) mm, size 805 x 170 x 120 mm, geometry from 6 cajas.STEP
          - object REF_RP_BOX45 at (995, 810, 599) mm, rotated rx 0 ry 0 rz 90 deg, size 400 x 170 x 120 mm, geometry from 3 cajas.STEP
        - folder LAYER 6
          - object REF_RP_BOX46 at (185, 810, 720) mm, rotated rx 0 ry 0 rz 90 deg, size 400 x 170 x 120 mm, geometry from 3 cajas.STEP
          - object REF_RP_BOX47 at (185, 0, 720) mm, rotated rx 0 ry 0 rz 90 deg, size 805 x 170 x 120 mm, geometry from 6 cajas.STEP
          - object REF_RP_BOX48 at (191, 0, 720) mm, size 805 x 170 x 120 mm, geometry from 6 cajas.STEP
          - object REF_RP_BOX49 at (191, 175, 720) mm, size 805 x 170 x 120 mm, geometry from 6 cajas.STEP
          - object REF_RP_BOX50 at (191, 350, 720) mm, size 805 x 170 x 120 mm, geometry from 6 cajas.STEP
          - object REF_RP_BOX51 at (191, 525, 720) mm, size 805 x 170 x 120 mm, geometry from 6 cajas.STEP
          - object REF_RP_BOX52 at (191, 700, 720) mm, size 805 x 170 x 120 mm, geometry from 6 cajas.STEP
          - object REF_RP_BOX53 at (191, 875, 720) mm, size 805 x 170 x 120 mm, geometry from 6 cajas.STEP
          - object REF_RP_BOX54 at (191, 1050, 720) mm, size 805 x 170 x 120 mm, geometry from 6 cajas.STEP
        - folder LAYER 7
          - object REF_RP_BOX55 at (995, 0, 841) mm, rotated rx 0 ry 0 rz 90 deg, size 805 x 170 x 120 mm, geometry from 6 cajas.STEP
          - object REF_RP_BOX56 at (15, 0, 841) mm, size 805 x 170 x 120 mm, geometry from 6 cajas.STEP
          - object REF_RP_BOX57 at (15, 175, 841) mm, size 805 x 170 x 120 mm, geometry from 6 cajas.STEP
          - object REF_RP_BOX58 at (15, 350, 841) mm, size 805 x 170 x 120 mm, geometry from 6 cajas.STEP
          - object REF_RP_BOX59 at (15, 525, 841) mm, size 805 x 170 x 120 mm, geometry from 6 cajas.STEP
          - object REF_RP_BOX60 at (15, 700, 841) mm, size 805 x 170 x 120 mm, geometry from 6 cajas.STEP
          - object REF_RP_BOX61 at (15, 875, 841) mm, size 805 x 170 x 120 mm, geometry from 6 cajas.STEP
          - object REF_RP_BOX62 at (15, 1050, 841) mm, size 805 x 170 x 120 mm, geometry from 6 cajas.STEP
          - object REF_RP_BOX63 at (995, 810, 841) mm, rotated rx 0 ry 0 rz 90 deg, size 400 x 170 x 120 mm, geometry from 3 cajas.STEP
        - folder LAYER 8
          - object REF_RP_BOX64 at (185, 810, 962) mm, rotated rx 0 ry 0 rz 90 deg, size 400 x 170 x 120 mm, geometry from 3 cajas.STEP
          - object REF_RP_BOX65 at (185, 0, 962) mm, rotated rx 0 ry 0 rz 90 deg, size 805 x 170 x 120 mm, geometry from 6 cajas.STEP
          - object REF_RP_BOX66 at (191, 0, 962) mm, size 805 x 170 x 120 mm, geometry from 6 cajas.STEP
          - object REF_RP_BOX67 at (191, 175, 962) mm, size 805 x 170 x 120 mm, geometry from 6 cajas.STEP
          - object REF_RP_BOX68 at (191, 350, 962) mm, size 805 x 170 x 120 mm, geometry from 6 cajas.STEP
          - object REF_RP_BOX69 at (191, 525, 962) mm, size 805 x 170 x 120 mm, geometry from 6 cajas.STEP
          - object REF_RP_BOX70 at (191, 700, 962) mm, size 805 x 170 x 120 mm, geometry from 6 cajas.STEP
          - object REF_RP_BOX71 at (191, 875, 962) mm, size 805 x 170 x 120 mm, geometry from 6 cajas.STEP
          - object REF_RP_BOX72 at (191, 1050, 962) mm, size 805 x 170 x 120 mm, geometry from 6 cajas.STEP
        - folder LAYER 9
          - object REF_RP_BOX73 at (995, 0, 1083) mm, rotated rx 0 ry 0 rz 90 deg, size 805 x 170 x 120 mm, geometry from 6 cajas.STEP
          - object REF_RP_BOX74 at (15, 0, 1083) mm, size 805 x 170 x 120 mm, geometry from 6 cajas.STEP
          - object REF_RP_BOX75 at (15, 175, 1083) mm, size 805 x 170 x 120 mm, geometry from 6 cajas.STEP
          - object REF_RP_BOX76 at (15, 350, 1083) mm, size 805 x 170 x 120 mm, geometry from 6 cajas.STEP
          - object REF_RP_BOX77 at (15, 525, 1083) mm, size 805 x 170 x 120 mm, geometry from 6 cajas.STEP
          - object REF_RP_BOX78 at (15, 700, 1083) mm, size 805 x 170 x 120 mm, geometry from 6 cajas.STEP
          - object REF_RP_BOX79 at (15, 875, 1083) mm, size 805 x 170 x 120 mm, geometry from 6 cajas.STEP
          - object REF_RP_BOX80 at (15, 1050, 1083) mm, size 805 x 170 x 120 mm, geometry from 6 cajas.STEP
          - object REF_RP_BOX81 at (995, 810, 1083) mm, rotated rx 0 ry 0 rz 90 deg, size 400 x 170 x 120 mm, geometry from 3 cajas.STEP
      - folder RP_Aux_Poses
        - target UP_RP (Cartesian target) at (765.99, 550.01, 1567.93) mm, rotated rx -179.99 ry 0 rz -90 deg; joints [-175.42, -8.86, 98.01, 0, 90.86, 94.58] of Doosan Robotics H2515
      - folder Place_RP
        - folder PL_LAYER 1
          - target RP_PL1 (Cartesian target) at (905, 402, 235) mm, rotated rx 180 ry 0 rz -90 deg; joints [-152.634, 94.466, 119.44, 0, -33.906, 117.366] of Doosan Robotics H2515
          - target RP_PL2 (Cartesian target) at (417, 80, 235) mm, rotated rx -180 ry 0 rz 0 deg; joints [-149.083, 90.04, 67.563, 0, 22.397, 30.917] of Doosan Robotics H2515
          - target RP_PL3 (Cartesian target) at (417, 255, 235) mm, rotated rx -180 ry 0 rz 0 deg; joints [-158.504, 88.046, 77.244, 0, 14.71, 21.496] of Doosan Robotics H2515
          - target RP_PL4 (Cartesian target) at (417, 430, 235) mm, rotated rx -180 ry 0 rz 0 deg; joints [-169.332, 87.219, 82.818, 0, 9.964, 10.668] of Doosan Robotics H2515
          - target RP_PL5 (Cartesian target) at (417, 605, 235) mm, rotated rx -180 ry 0 rz 0 deg; joints [-181.006, 87.015, 84.586, 0, 8.399, -1.006] of Doosan Robotics H2515
          - target RP_PL6 (Cartesian target) at (417, 780, 235) mm, rotated rx -180 ry 0 rz 0 deg; joints [-192.624, 87.245, 82.603, 0, 10.152, -12.624] of Doosan Robotics H2515
          - target RP_PL7 (Cartesian target) at (417, 955, 235) mm, rotated rx -180 ry 0 rz 0 deg; joints [-203.308, 88.122, 76.806, 0, 15.072, -23.308] of Doosan Robotics H2515
          - target RP_PL8 (Cartesian target) at (417, 1130, 235) mm, rotated rx -180 ry 0 rz 0 deg; joints [-212.542, 90.206, 66.87, 0, 22.924, -32.542] of Doosan Robotics H2515
          - target RP_PL9 (Cartesian target) at (905, 1213, 235) mm, rotated rx 180 ry 0 rz -90 deg; joints [-240.303, 86.647, 97.692, 0, -4.339, 29.697] of Doosan Robotics H2515
        - folder PL_LAYER 2
          - target RP_PL10 (Cartesian target) at (95, 808, 356) mm, rotated rx -180 ry 0 rz -90 deg; joints [-190.549, 90.465, 45.603, 0, 43.932, 79.451] of Doosan Robotics H2515
          - target RP_PL11 (Cartesian target) at (95, 402, 356) mm, rotated rx 180 ry 0 rz -90 deg; joints [-170.88, 90.34, 45.948, 0, 43.712, 99.12] of Doosan Robotics H2515
          - target RP_PL12 (Cartesian target) at (593, 80, 356) mm, rotated rx 180 ry 0 rz 0 deg; joints [-142.975, 78.008, 91.998, 0, 9.993, 37.025] of Doosan Robotics H2515
          - target RP_PL13 (Cartesian target) at (593, 255, 356) mm, rotated rx -180 ry 0 rz 0 deg; joints [-153.609, 77.297, 101.288, 0, 1.415, 26.391] of Doosan Robotics H2515
          - target RP_PL14 (Cartesian target) at (593, 430, 356) mm, rotated rx -180 ry 0 rz 0 deg; joints [-166.641, 77.422, 106.948, 0, -4.37, 13.359] of Doosan Robotics H2515
          - target RP_PL15 (Cartesian target) at (593, 605, 356) mm, rotated rx -180 ry 0 rz 0 deg; joints [-181.269, 77.578, 108.796, 0, -6.374, -1.269] of Doosan Robotics H2515
          - target RP_PL16 (Cartesian target) at (593, 780, 356) mm, rotated rx -180 ry 0 rz 0 deg; joints [-195.788, 77.407, 106.726, 0, -4.133, -15.788] of Doosan Robotics H2515
          - target RP_PL17 (Cartesian target) at (593, 955, 356) mm, rotated rx 180 ry 0 rz 0 deg; joints [-208.557, 77.307, 100.853, 0, 1.84, -28.557] of Doosan Robotics H2515
          - target RP_PL18 (Cartesian target) at (593, 1130, 356) mm, rotated rx -180 ry 0 rz 0 deg; joints [-218.883, 78.091, 91.359, 0, 10.55, -38.883] of Doosan Robotics H2515
        - folder PL_LAYER 3
          - target RP_PL19 (Cartesian target) at (905, 402, 477) mm, rotated rx -180 ry 0 rz -90 deg; joints [-152.634, 74.873, 136.398, 0, -31.27, 117.366] of Doosan Robotics H2515
          - target RP_PL20 (Cartesian target) at (417, 80, 477) mm, rotated rx -180 ry 0 rz 0 deg; joints [-149.083, 72.685, 81.429, 0, 25.886, 30.917] of Doosan Robotics H2515
          - target RP_PL21 (Cartesian target) at (417, 255, 477) mm, rotated rx -180 ry 0 rz 0 deg; joints [-158.504, 70.403, 90.678, 0, 18.919, 21.496] of Doosan Robotics H2515
          - target RP_PL22 (Cartesian target) at (417, 430, 477) mm, rotated rx -180 ry 0 rz 0 deg; joints [-169.332, 69.304, 96.177, 0, 14.519, 10.668] of Doosan Robotics H2515
          - target RP_PL23 (Cartesian target) at (417, 605, 477) mm, rotated rx -180 ry 0 rz 0 deg; joints [-181.006, 68.999, 97.949, 0, 13.052, -1.006] of Doosan Robotics H2515
          - target RP_PL24 (Cartesian target) at (417, 780, 477) mm, rotated rx -180 ry 0 rz 0 deg; joints [-192.624, 69.342, 95.963, 0, 14.695, -12.624] of Doosan Robotics H2515
          - target RP_PL25 (Cartesian target) at (417, 955, 477) mm, rotated rx -180 ry 0 rz 0 deg; joints [-203.308, 70.497, 90.252, 0, 19.251, -23.308] of Doosan Robotics H2515
          - target RP_PL26 (Cartesian target) at (417, 1130, 477) mm, rotated rx -180 ry 0 rz 0 deg; joints [-212.542, 72.862, 80.782, 0, 26.356, -32.542] of Doosan Robotics H2515
          - target RP_PL27 (Cartesian target) at (905, 1213, 477) mm, rotated rx -180 ry 0 rz -90 deg; joints [-240.303, 67.705, 111.499, 0, 0.796, 29.697] of Doosan Robotics H2515
        - folder PL_LAYER 4
          - target RP_PL28 (Cartesian target) at (95, 808, 598) mm, rotated rx -180 ry 0 rz -90 deg; joints [-190.549, 74.228, 58.047, 0, 47.725, 79.451] of Doosan Robotics H2515
          - target RP_PL29 (Cartesian target) at (95, 402, 598) mm, rotated rx -180 ry 0 rz -90 deg; joints [-170.88, 74.116, 58.338, 0, 47.546, 99.12] of Doosan Robotics H2515
          - target RP_PL30 (Cartesian target) at (593, 80, 598) mm, rotated rx -180 ry 0 rz 0 deg; joints [-142.975, 60.094, 101.845, 0, 18.061, 37.025] of Doosan Robotics H2515
          - target RP_PL31 (Cartesian target) at (593, 255, 598) mm, rotated rx 180 ry 0 rz 0 deg; joints [-153.609, 58.28, 111.477, 0, 10.243, 26.391] of Doosan Robotics H2515
          - target RP_PL32 (Cartesian target) at (593, 430, 598) mm, rotated rx -180 ry 0 rz 0 deg; joints [-166.641, 57.601, 117.51, 0, 4.889, 13.359] of Doosan Robotics H2515
          - target RP_PL33 (Cartesian target) at (593, 605, 598) mm, rotated rx -180 ry 0 rz 0 deg; joints [-181.269, 57.476, 119.511, 0, 3.013, -1.269] of Doosan Robotics H2515
          - target RP_PL34 (Cartesian target) at (593, 780, 598) mm, rotated rx -180 ry 0 rz 0 deg; joints [-195.788, 57.62, 117.27, 0, 5.11, -15.788] of Doosan Robotics H2515
          - target RP_PL35 (Cartesian target) at (593, 955, 598) mm, rotated rx -180 ry 0 rz 0 deg; joints [-208.557, 58.347, 111.02, 0, 10.633, -28.557] of Doosan Robotics H2515
          - target RP_PL36 (Cartesian target) at (593, 1130, 598) mm, rotated rx -180 ry 0 rz 0 deg; joints [-218.883, 60.242, 101.193, 0, 18.565, -38.883] of Doosan Robotics H2515
      - folder Waypoints_RP
        - target MID_RP_L1 (Cartesian target) at (500, 605, 600) mm, rotated rx -180 ry 0 rz 0 deg; joints [-181.114, 58.267, 110.565, 0, 11.168, -1.114] of Doosan Robotics H2515
        - target MID_RP_L2 (Cartesian target) at (500, 605, 721) mm, rotated rx -180 ry 0 rz 0 deg; joints [-181.114, 48.753, 112.909, 0, 18.337, -1.114] of Doosan Robotics H2515
        - target MID_RP_L3 (Cartesian target) at (500, 605, 842) mm, rotated rx -180 ry 0 rz 0 deg; joints [-181.114, 39.587, 113.339, 0, 27.074, -1.114] of Doosan Robotics H2515
        - target MID_RP_L4 (Cartesian target) at (500, 605, 962) mm, rotated rx -180 ry 0 rz 0 deg; joints [-181.114, 31.262, 111.856, 0, 36.882, -1.114] of Doosan Robotics H2515
        - target MID_RP_L5 (Cartesian target) at (500, 605, 1082) mm, rotated rx -180 ry 0 rz 0 deg; joints [-181.114, 24.104, 108.528, 0, 47.368, -1.114] of Doosan Robotics H2515
    - frame Lift100_Frame at (0, 0, 0) mm
      - object Lift100 at (0, 0, 0) mm, size 565.7 x 561 x 747.5 mm, geometry from Lift100.STEP
  - folder Auxiliar Programs
  - folder Python
    - Python program Export_Pallet_Positions (listed below)
  - folder Test
    - program Prog1 (38 instructions, listed below)
  - Python program crear_places (listed below)
  - Python program crear_app (listed below)
  - Python program crear_reccorido (listed below)
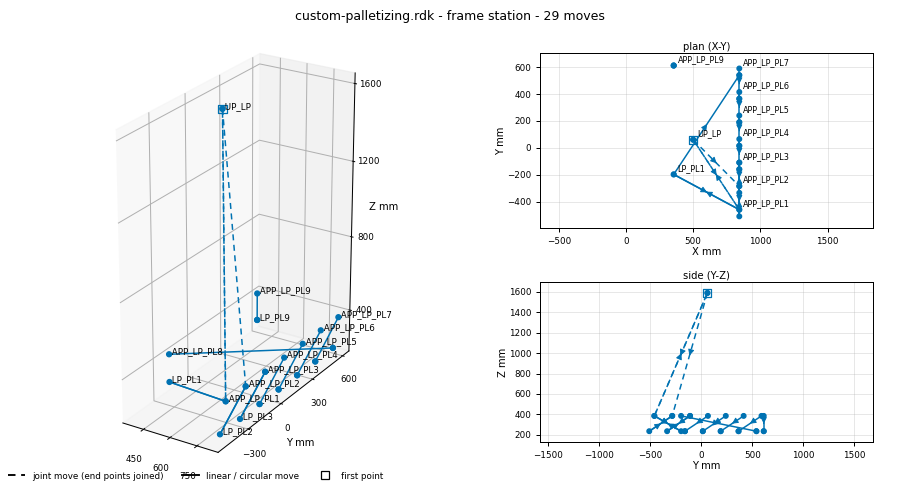
[picture p0: tool path of custom-palletizing.rdk in frame station, 29 of 36 moves have a stored position in this frame; points joined in program order, loops and branches not executed]

--- Python program Export_Pallet_Positions ---
# Exporta solo PLACE en cartesiano (TCP respecto a un frame)
# Autor: Mario Padilla

from robodk import robolink as RL
from robodk import robomath as rdk
import os
from datetime import datetime

RDK = RL.Robolink()

# ========= CONFIGURACIÓN =========
# Nombre del frame de referencia (el TCP se expresará respecto a este frame)
REF_FRAME_NAME = 'Left_Pallet_Frame'

# Nombres de las carpetas (tal como aparecen en el Árbol de RoboDK)
# Ejemplo de rutas (de hijo a raíz):
#   PLACE:  PL_LAYER 9   ->  Place_LP   ->  Left_Pallet_Frame
PL_LAYER_NAME  = 'PL_LAYER 9'
PLACE_PARENT   = 'Place_LP'

# ========= UTILIDADES =========
def wrap_deg(a):
    """Normaliza ángulos a (-180, 180]."""
    a = (a + 180.0) % 360.0 - 180.0
    return 0.0 if abs(a) < 1e-9 else a

def has_ancestor_path(item, path_child_to_root):
    """¿El item pertenece a la ruta (de hijo a raíz) dada por nombres?"""
    idx = 0
    p = item.Parent()
    while p.Valid() and idx < len(path_child_to_root):
        if p.Name() == path_child_to_root[idx]:
            idx += 1
        p = p.Parent()
    return idx == len(path_child_to_root)

def pose_rel_and_abs(target, H_ref_abs):
    """Devuelve (H_rel, H_abs): TCP vs Ref y TCP vs Mundo."""
    H_abs = target.PoseAbs()             # pose absoluta del target (TCP vs World)
    H_rel = rdk.invH(H_ref_abs) * H_abs  # relativa al frame de referencia
    return H_rel, H_abs

def TxyzRxyz_deg(H_rel):
    """Convierte una pose a (X,Y,Z,Rx,Ry,Rz) con grados tipo panel."""
    x, y, z, rx, ry, rz = rdk.Pose_2_TxyzRxyz(H_rel)  # rx,ry,rz en rad
    todeg = 180.0 / rdk.pi
    rx, ry, rz = rx*todeg, ry*todeg, rz*todeg
    # Ajuste de signo en Rz para coincidir con el panel de RoboDK (Adept/Comau/Kawasaki):
    rz = -rz
    return x, y, z, wrap_deg(rx), wrap_deg(ry), wrap_deg(rz)

# ========= FRAME =========
ref_frame = RDK.Item(REF_FRAME_NAME, RL.ITEM_TYPE_FRAME)
if not ref_frame.Valid():
    RDK.ShowMessage(f'❌ No se encontró el frame "{REF_FRAME_NAME}"')
    raise SystemExit
H_ref_abs = ref_frame.PoseAbs()

# ========= RECOLECCIÓN DE TARGETS =========
all_targets = RDK.ItemList(RL.ITEM_TYPE_TARGET)

# ruta de hijo→raíz
PLACE_PATH_CHILD_TO_ROOT = [PL_LAYER_NAME, PLACE_PARENT, REF_FRAME_NAME]

places = [t for t in all_targets if has_ancestor_path(t, PLACE_PATH_CHILD_TO_ROOT)]

if not places:
    RDK.ShowMessage('❌ No se encontraron targets de PLACE en la ruta indicada')
    raise SystemExit

# ordenados por nombre
places.sort(key=lambda i: i.Name())

# ========= GENERACIÓN DE TEXTO =========
lines = []
lines.append(f'Frame de referencia: "{REF_FRAME_NAME}"\n\n')
lines.append(f'== PLACE: {PLACE_PARENT} / {PL_LAYER_NAME} ==\n')
lines.append('Nombre (X(mm), Y(mm), Z(mm), Rx(deg), Ry(deg), Rz(deg))\n')

for t in places:
    H_rel, _ = pose_rel_and_abs(t, H_ref_abs)
    x, y, z, rx, ry, rz = TxyzRxyz_deg(H_rel)
    line = f'{t.Name()} ( {round(x,3)}, {round(y,3)}, {round(z,3)}, {round(rx,3)}, {round(ry,3)}, {round(rz,3)} )'
    lines.append(line + '\n')

# ========= GUARDAR EN ESCRITORIO =========
desktop = os.path.join(os.path.expanduser('~'), 'Desktop')
ts = datetime.now().strftime('%Y-%m-%d_%H-%M-%S')
filepath = os.path.join(desktop, f'Pallet_PLACE_Targets_{ts}.txt')

with open(filepath, 'w', encoding='utf-8') as f:
    f.writelines(lines)

RDK.ShowMessage(f'✅ Archivo exportado en:\n{filepath}')

--- program Prog1 (robot Doosan Robotics H2515) ---
  Est. Ref.: Left_Pallet_Frame
  Est. herr: Gripper
  MoveJ (UP_LP)
  MoveJ (APP_LP_PL1)
  MoveL (LP_PL1)
  MoveL (APP_LP_PL1)
  MoveJ (UP_LP)
  MoveJ (APP_LP_PL2)
  MoveL (LP_PL2)
  MoveL (APP_LP_PL2)
  MoveJ (UP_LP) [its target is no longer in the station]
  MoveJ (APP_LP_PL3)
  MoveL (LP_PL3)
  MoveL (APP_LP_PL3)
  MoveJ (UP_LP) [its target is no longer in the station]
  MoveJ (APP_LP_PL4)
  MoveL (LP_PL4)
  MoveL (LP_PL4)
  MoveJ (UP_LP) [its target is no longer in the station]
  MoveJ (APP_LP_PL5)
  MoveL (LP_PL5)
  MoveL (LP_PL5)
  MoveJ (UP_LP) [its target is no longer in the station]
  MoveJ (APP_LP_PL6)
  MoveL (LP_PL6)
  MoveL (LP_PL6)
  MoveJ (UP_LP) [its target is no longer in the station]
  MoveJ (APP_LP_PL7)
  MoveL (LP_PL7)
  MoveL (LP_PL7)
  MoveJ (UP_LP) [its target is no longer in the station]
  MoveJ (APP_LP_PL8)
  MoveL (LP_PL8)
  MoveL (LP_PL8)
  MoveJ (UP_LP) [its target is no longer in the station]
  MoveJ (APP_LP_PL9)
  MoveL (LP_PL9)
  MoveL (LP_PL9)

--- Python program crear_places ---
from robodk import robolink, robomath

RDK = robolink.Robolink()

# Parámetros
place_lp = RDK.Item('Place_LP', robolink.ITEM_TYPE_FOLDER)
z_increment = 120  # mm por capa
num_layers = 9
positions_per_layer = 9  # LP_PL1-9, LP_PL10-18, etc.

# Capas base
layer1 = RDK.Item('PL_LAYER 1', robolink.ITEM_TYPE_FOLDER)
layer2 = RDK.Item('PL_LAYER 2', robolink.ITEM_TYPE_FOLDER)

# Obtener targets base
targets_layer1 = [t for t in layer1.Childs() if t.Type() == robolink.ITEM_TYPE_TARGET]
targets_layer2 = [t for t in layer2.Childs() if t.Type() == robolink.ITEM_TYPE_TARGET]

# Contador global: Layer 3 empieza en LP_PL19
count = 18

# Iterar sobre las capas 3 a 9
for layer_idx in range(3, num_layers + 1):
    # Alternar capa base
    base_targets = targets_layer1 if layer_idx % 2 == 1 else targets_layer2

    # Buscar carpeta existente
    layer_folder_name = f'PL_LAYER {layer_idx}'
    new_layer_folder = None
    for child in place_lp.Childs():
        if child.Name() == layer_folder_name:
            new_layer_folder = child
            break

    if new_layer_folder is None or not new_layer_folder.Valid():
        raise Exception(f"No se encontró la carpeta {layer_folder_name}")

    # Offset acumulado en Z hacia arriba
    if layer_idx % 2 == 1:
        offset_z = (layer_idx) * z_increment  # Layer 3 = 240 mm
        offset_vector = robomath.transl(0, 0, -offset_z)
    else:
        offset_z = (layer_idx-1) * z_increment  # Define offset_z for even layers as well
        offset_vector = robomath.transl(0, 0, -offset_z)

    print(f"este es el layer: {layer_idx}")
    # Si actualmente baja, invertimos
     # positivo hacia arriba
    print(f"este es el vector: {offset_vector}")


        # Crear targets dentro de la carpeta
    for t in base_targets:
        count += 1
        new_name = f'LP_PL{count}'

        # Pose con offset
        pose = t.Pose() * offset_vector
        ref_frame = t.Parent()
        tool = t.getLink(robolink.ITEM_TYPE_TOOL)

        # Crear target dentro de la carpeta existente
        new_target = RDK.AddTarget(new_name, new_layer_folder, ref_frame)
        new_target.setPose(pose)
        if tool.Valid():
            new_target.setTool(tool)

print("✅ Posiciones agregadas correctamente a las carpetas existentes con offset Z hacia arriba y numeración desde LP_PL19.")

--- Python program crear_app ---
from robodk import robolink, robomath

RDK = robolink.Robolink()

# Parámetros
place_lp = RDK.Item('App_PL_LP', robolink.ITEM_TYPE_FOLDER)
z_increment = 150  # mm por capa
num_layers = 9
positions_per_layer = 9

# Capas base
layer1 = RDK.Item('APP_LAYER 1', robolink.ITEM_TYPE_FOLDER)
layer2 = RDK.Item('APP_LAYER 2', robolink.ITEM_TYPE_FOLDER)

# Obtener targets base
targets_layer1 = [t for t in layer1.Childs() if t.Type() == robolink.ITEM_TYPE_TARGET]
targets_layer2 = [t for t in layer2.Childs() if t.Type() == robolink.ITEM_TYPE_TARGET]
count = 18

# Iterar sobre las capas 3 a 9
for layer_idx in range(3, num_layers + 1):
    base_targets = targets_layer1 if layer_idx % 2 == 1 else targets_layer2

    layer_folder_name = f'APP_LAYER {layer_idx}'
    new_layer_folder = None
    for child in place_lp.Childs():
        if child.Name() == layer_folder_name:
            new_layer_folder = child
            break

    if new_layer_folder is None or not new_layer_folder.Valid():
        raise Exception(f"No se encontró la carpeta {layer_folder_name}")

    # Offset acumulado en Z hacia arriba
    if layer_idx % 2 == 1:
        offset_z = (layer_idx) * z_increment  # Layer 3 = 240 mm
        offset_vector = robomath.transl(0, 0, -offset_z)
    else:
        offset_z = (layer_idx-1) * z_increment  # Define offset_z for even layers as well
        offset_vector = robomath.transl(0, 0, -offset_z)

    print(f"este es el layer: {layer_idx}")
    print(f"este es el vector: {offset_vector}")


        # Crear targets dentro de la carpeta
    for t in base_targets:
        count += 1
        new_name = f'APP_LP_PL{count}'

        # Pose con offset
        pose = t.Pose() * offset_vector
        ref_frame = t.Parent()
        tool = t.getLink(robolink.ITEM_TYPE_TOOL)

        # Crear target dentro de la carpeta existente
        new_target = RDK.AddTarget(new_name, new_layer_folder, ref_frame)
        new_target.setPose(pose)
        if tool.Valid():
            new_target.setTool(tool)

print("✅ Posiciones agregadas correctamente a las carpetas existentes con offset Z hacia arriba y numeración desde APP_LP_PL19.")

--- Python program crear_reccorido ---
from robodk import robolink

RDK = robolink.Robolink()

print("Lista de items en la estación:")
for item in RDK.ItemList():
    print(item.Name(), item.Type())
